FUNCTION_BLOCK RtdReadings

VAR
	Rtd01 : FB_Pt100;
	Rtd02 : FB_Pt100;
	Rtd03 : FB_Pt100;
	Rtd04 : FB_Pt100;
	Rtd05 : FB_Pt100;
	Rtd06 : FB_Pt100;
END_VAR

//Instances of PT100, temperature measurement
Rtd01(Raw := IO.TBL_RTD01_TEMP,TempFaranheit =>G_Epics.RtdTemperature.TBL_RTD01_TEMP);
Rtd02(Raw := IO.TBL_RTD02_TEMP,TempFaranheit =>G_Epics.RtdTemperature.TBL_RTD02_TEMP);
Rtd03(Raw := IO.TBL_RTD03_TEMP,TempFaranheit =>G_Epics.RtdTemperature.TBL_RTD03_TEMP);
Rtd04(Raw := IO.TBL_RTD04_TEMP,TempFaranheit =>G_Epics.RtdTemperature.TBL_RTD04_TEMP);
Rtd05(Raw := IO.TBL_RTD05_TEMP,TempFaranheit =>G_Epics.RtdTemperature.TBL_RTD05_TEMP);
Rtd06(Raw := IO.TBL_RTD06_TEMP,TempFaranheit =>G_Epics.RtdTemperature.TBL_RTD06_TEMP);

END_FUNCTION_BLOCK

(* stored: Version 1.1.0.1, ProductVersion 3.1.4024.9
   POU RtdReadings: Id {c7d6eca6-3114-48f2-ade9-4d051967e7a0}, SpecialFunc None *)
